// TIA Portal V19 export
FUNCTION_BLOCK "ValveMonitor"   // FB2, STL
TITLE = Valve Monitor
{ S7_Optimized_Access := 'TRUE' }
// Valve Monitor monitors single acting valves with Energiseed only or 
// De-energised 
// only or both Feedback states. Selection of feedback states in use can be 
// selected with Bits 0 and 1 of the "ControlWord" Input.
// 
// 
// Control Word
// Bit 0 = IN_DE in use
// Bit 1 = IN_EN in use
// 
// 
// Valve Monitor should be called within a Timed Interrupt OB and the duration 
// counters should be multiplied by the Timed Interrupt Cycle time to get the 
// durations in Seconds.
// 
// Note: If Activation State changes before destination FeedBack is reached then 
// the Duration count is not moved to the Archive and therefore does not affect 
// the 
// average duration. (De)Activations Count(s) will be incremented
// stored: AutoNumber false, MemoryReserve 100
   VAR_INPUT
      IN_EN : Bool;
      IN_DE : Bool;
      IN_ACT : Bool;
      ControlWord : Word;
   END_VAR
   VAR_IN_OUT
      Info : "ValvesInfo_UDT";
   END_VAR
   VAR
      ActMem : Bool;
      DeActMem : Bool;
      ActDur : Bool;
      DeActDur : Bool;
      ActClearDurCount : Bool;
      DeActClearDurCount : Bool;
      FP_A : Bool;
      FP_D : Bool;
      FP_A_Pulse : Bool;
      FP_D_Pulse : Bool;
      SumAverage : DInt;
      CountAverage : Int;
      data : "ValveMonitor_UDT";
   END_VAR
   VAR_TEMP
      EN_In_Use : Bool;
      DE_In_Use : Bool;
   END_VAR
BEGIN

NETWORK
TITLE = 
      A     #ControlWord.%X0;
      =     #EN_In_Use;
      A     #ControlWord.%X1;
      =     #DE_In_Use;


NETWORK
TITLE = RESET ALL Info
      A     #Info.RESET;
      JCN   RST;
      L     0;
// Act
      T     #data.Activation.ActivationCounter;
      T     #data.Activation.StrokeDuration.count;
      T     #data.Activation.StrokeDuration.Archive.n1;
      T     #data.Activation.StrokeDuration.Archive.n2;
      T     #data.Activation.StrokeDuration.Archive.n3;
      T     #data.Activation.StrokeDuration.Archive.n4;
      T     #data.Activation.StrokeDuration.Archive.n5;
      T     #data.Activation.StrokeDuration.Archive.n6;
      T     #data.Activation.StrokeDuration.Archive.n7;
      T     #data.Activation.StrokeDuration.Archive.n8;
      T     #data.Activation.StrokeDuration.Archive.n9;
      T     #data.Activation.StrokeDuration.Archive.n10;
// De_Act
      T     #data.De_Activation.De_ActivationCounter;
      T     #data.De_Activation.StrokeDuration.count;
      T     #data.De_Activation.StrokeDuration.Archive.n1;
      T     #data.De_Activation.StrokeDuration.Archive.n2;
      T     #data.De_Activation.StrokeDuration.Archive.n3;
      T     #data.De_Activation.StrokeDuration.Archive.n4;
      T     #data.De_Activation.StrokeDuration.Archive.n5;
      T     #data.De_Activation.StrokeDuration.Archive.n6;
      T     #data.De_Activation.StrokeDuration.Archive.n7;
      T     #data.De_Activation.StrokeDuration.Archive.n8;
      T     #data.De_Activation.StrokeDuration.Archive.n9;
      T     #data.De_Activation.StrokeDuration.Archive.n10;
      R     #Info.RESET;
RST:  NOP   0;


NETWORK
TITLE = Activation Counter
      A     #IN_ACT;
      AN    #IN_EN;
      AN    #ActMem;
      S     #ActMem;
      R     #DeActMem;

      A     #ActMem;
      FP    #FP_A;
      =     #FP_A_Pulse;
      JCN   ACTC;
      L     #data.Activation.ActivationCounter;
      L     1;
      +I;
      T     #data.Activation.ActivationCounter;
ACTC: NOP   0;


NETWORK
TITLE = De-Activation Counter
      AN    #IN_ACT;
      AN    #IN_DE;
      AN    #DeActMem;
      S     #DeActMem;
      R     #ActMem;

      A     #DeActMem;
      FP    #FP_D;
      =     #FP_D_Pulse;
      JCN   DACC;
      L     #data.De_Activation.De_ActivationCounter;
      L     1;
      +I;
      T     #data.De_Activation.De_ActivationCounter;
DACC: NOP   0;



NETWORK
TITLE = Activation Duration
      A     #EN_In_Use;  // IN_EN in Use
      JCN   ENDA;  // Jump to ENDA if False
      A     #FP_A_Pulse;
      AN    #IN_EN;
      S     #ActDur;

      A     #ActDur;
      A     #IN_EN;
      ON    #IN_ACT;
      R     #ActDur;
      R     #ActClearDurCount;
// Move Duration Count to Archive.n1
      AN    #ActDur;
      A     #IN_ACT;
      JCN   MOV;
      L     #data.Activation.StrokeDuration.count;
      T     #data.Activation.StrokeDuration.Archive.n1;
MOV:  NOP   0;

//Clear Counter
      A     #ActDur;
      AN    #ActClearDurCount;
      JCN   ATCC;
      L     0;
      T     #data.Activation.StrokeDuration.count;
      SET;
      S     #ActClearDurCount;
// Shift Archive data
      L     #data.Activation.StrokeDuration.Archive.n9;
      T     #data.Activation.StrokeDuration.Archive.n10;
      L     #data.Activation.StrokeDuration.Archive.n8;
      T     #data.Activation.StrokeDuration.Archive.n9;
      L     #data.Activation.StrokeDuration.Archive.n7;
      T     #data.Activation.StrokeDuration.Archive.n8;
      L     #data.Activation.StrokeDuration.Archive.n6;
      T     #data.Activation.StrokeDuration.Archive.n7;
      L     #data.Activation.StrokeDuration.Archive.n5;
      T     #data.Activation.StrokeDuration.Archive.n6;
      L     #data.Activation.StrokeDuration.Archive.n4;
      T     #data.Activation.StrokeDuration.Archive.n5;
      L     #data.Activation.StrokeDuration.Archive.n3;
      T     #data.Activation.StrokeDuration.Archive.n4;
      L     #data.Activation.StrokeDuration.Archive.n2;
      T     #data.Activation.StrokeDuration.Archive.n3;
      L     #data.Activation.StrokeDuration.Archive.n1;
      T     #data.Activation.StrokeDuration.Archive.n2;
ATCC: NOP   0;

// Count Duration
      A     #ActDur;
      A     #ActClearDurCount;
      JCN   _0CD;
      L     #data.Activation.StrokeDuration.count;
      L     1;
      +I;
      T     #data.Activation.StrokeDuration.count;
_0CD: NOP   0;
ENDA: NOP   0;




NETWORK
TITLE = DeDeActivation Duration
      A     #DE_In_Use;  // IN_DE in Use
      JCN   ENDD;  // Jump to ENDA if False
      A     #FP_D_Pulse;
      AN    #IN_DE;
      S     #DeActDur;

      A     #DeActDur;
      A     #IN_DE;
      O     #IN_ACT;
      R     #DeActDur;
      R     #DeActClearDurCount;
// Move Duration Count to Archive.n1
      AN    #DeActDur;
      AN    #IN_ACT;
      JCN   MOVD;
      L     #data.De_Activation.StrokeDuration.count;
      T     #data.De_Activation.StrokeDuration.Archive.n1;
MOVD: NOP   0;

//Clear Counter
      A     #DeActDur;
      AN    #DeActClearDurCount;
      JCN   DTCC;
      L     0;
      T     #data.De_Activation.StrokeDuration.count;
      SET;
      S     #DeActClearDurCount;
// Shift Archive data
      L     #data.De_Activation.StrokeDuration.Archive.n9;
      T     #data.De_Activation.StrokeDuration.Archive.n10;
      L     #data.De_Activation.StrokeDuration.Archive.n8;
      T     #data.De_Activation.StrokeDuration.Archive.n9;
      L     #data.De_Activation.StrokeDuration.Archive.n7;
      T     #data.De_Activation.StrokeDuration.Archive.n8;
      L     #data.De_Activation.StrokeDuration.Archive.n6;
      T     #data.De_Activation.StrokeDuration.Archive.n7;
      L     #data.De_Activation.StrokeDuration.Archive.n5;
      T     #data.De_Activation.StrokeDuration.Archive.n6;
      L     #data.De_Activation.StrokeDuration.Archive.n4;
      T     #data.De_Activation.StrokeDuration.Archive.n5;
      L     #data.De_Activation.StrokeDuration.Archive.n3;
      T     #data.De_Activation.StrokeDuration.Archive.n4;
      L     #data.De_Activation.StrokeDuration.Archive.n2;
      T     #data.De_Activation.StrokeDuration.Archive.n3;
      L     #data.De_Activation.StrokeDuration.Archive.n1;
      T     #data.De_Activation.StrokeDuration.Archive.n2;
DTCC: NOP   0;

// Count Duration
      A     #DeActDur;
      A     #DeActClearDurCount;
      JCN   D0CD;
      L     #data.De_Activation.StrokeDuration.count;
      L     1;
      +I;
      T     #data.De_Activation.StrokeDuration.count;
D0CD: NOP   0;
ENDD: NOP   0;




NETWORK
TITLE = Average Activation Duration Count
      L     0;
      T     #SumAverage;
      T     #CountAverage;


      L     #data.Activation.StrokeDuration.Archive.n1;
      L     0;
      >I;
      JCN   a001;
      L     1;
      L     #CountAverage;
      +I;
      T     #CountAverage;
      L     #data.Activation.StrokeDuration.Archive.n1;
      L     #SumAverage;
      +I;
      T     #SumAverage;
a001: L     #data.Activation.StrokeDuration.Archive.n2;
      L     0;
      >I;
      JCN   a002;
      L     1;
      L     #CountAverage;
      +I;
      T     #CountAverage;
      L     #data.Activation.StrokeDuration.Archive.n2;
      L     #SumAverage;
      +I;
      T     #SumAverage;
a002: L     #data.Activation.StrokeDuration.Archive.n3;
      L     0;
      >I;
      JCN   a003;
      L     1;
      L     #CountAverage;
      +I;
      T     #CountAverage;
      L     #data.Activation.StrokeDuration.Archive.n3;
      L     #SumAverage;
      +I;
      T     #SumAverage;
a003: L     #data.Activation.StrokeDuration.Archive.n4;
      L     0;
      >I;
      JCN   a004;
      L     1;
      L     #CountAverage;
      +I;
      T     #CountAverage;
      L     #data.Activation.StrokeDuration.Archive.n4;
      L     #SumAverage;
      +I;
      T     #SumAverage;
a004: L     #data.Activation.StrokeDuration.Archive.n5;
      L     0;
      >I;
      JCN   a005;
      L     1;
      L     #CountAverage;
      +I;
      T     #CountAverage;
      L     #data.Activation.StrokeDuration.Archive.n5;
      L     #SumAverage;
      +I;
      T     #SumAverage;
a005: L     #data.Activation.StrokeDuration.Archive.n6;
      L     0;
      >I;
      JCN   a006;
      L     1;
      L     #CountAverage;
      +I;
      T     #CountAverage;
      L     #data.Activation.StrokeDuration.Archive.n6;
      L     #SumAverage;
      +I;
      T     #SumAverage;
a006: L     #data.Activation.StrokeDuration.Archive.n7;
      L     0;
      >I;
      JCN   a007;
      L     1;
      L     #CountAverage;
      +I;
      T     #CountAverage;
      L     #data.Activation.StrokeDuration.Archive.n7;
      L     #SumAverage;
      +I;
      T     #SumAverage;
a007: L     #data.Activation.StrokeDuration.Archive.n8;
      L     0;
      >I;
      JCN   a008;
      L     1;
      L     #CountAverage;
      +I;
      T     #CountAverage;
      L     #data.Activation.StrokeDuration.Archive.n8;
      L     #SumAverage;
      +I;
      T     #SumAverage;
a008: L     #data.Activation.StrokeDuration.Archive.n9;
      L     0;
      >I;
      JCN   a009;
      L     1;
      L     #CountAverage;
      +I;
      T     #CountAverage;
      L     #data.Activation.StrokeDuration.Archive.n9;
      L     #SumAverage;
      +I;
      T     #SumAverage;
a009: L     #data.Activation.StrokeDuration.Archive.n10;
      L     0;
      >I;
      JCN   a010;
      L     1;
      L     #CountAverage;
      +I;
      T     #CountAverage;
      L     #data.Activation.StrokeDuration.Archive.n10;
      L     #SumAverage;
      +I;
      T     #SumAverage;
a010: NOP   0;
// Calculate Average
      L     #SumAverage;
      L     #CountAverage;
      /D;
      T     #data.Activation.StrokeDuration.Average;


NETWORK
TITLE = Average De_Activation Duration Count
      L     0;
      T     #SumAverage;
      T     #CountAverage;


      L     #data.Activation.StrokeDuration.Archive.n1;
      L     0;
      >I;
      JCN   d001;
      L     1;
      L     #CountAverage;
      +I;
      T     #CountAverage;
      L     #data.De_Activation.StrokeDuration.Archive.n1;
      L     #SumAverage;
      +I;
      T     #SumAverage;
d001: L     #data.De_Activation.StrokeDuration.Archive.n2;
      L     0;
      >I;
      JCN   d002;
      L     1;
      L     #CountAverage;
      +I;
      T     #CountAverage;
      L     #data.De_Activation.StrokeDuration.Archive.n2;
      L     #SumAverage;
      +I;
      T     #SumAverage;
d002: L     #data.De_Activation.StrokeDuration.Archive.n3;
      L     0;
      >I;
      JCN   d003;
      L     1;
      L     #CountAverage;
      +I;
      T     #CountAverage;
      L     #data.De_Activation.StrokeDuration.Archive.n3;
      L     #SumAverage;
      +I;
      T     #SumAverage;
d003: L     #data.De_Activation.StrokeDuration.Archive.n4;
      L     0;
      >I;
      JCN   d004;
      L     1;
      L     #CountAverage;
      +I;
      T     #CountAverage;
      L     #data.De_Activation.StrokeDuration.Archive.n4;
      L     #SumAverage;
      +I;
      T     #SumAverage;
d004: L     #data.De_Activation.StrokeDuration.Archive.n5;
      L     0;
      >I;
      JCN   d005;
      L     1;
      L     #CountAverage;
      +I;
      T     #CountAverage;
      L     #data.De_Activation.StrokeDuration.Archive.n5;
      L     #SumAverage;
      +I;
      T     #SumAverage;
d005: L     #data.De_Activation.StrokeDuration.Archive.n6;
      L     0;
      >I;
      JCN   d006;
      L     1;
      L     #CountAverage;
      +I;
      T     #CountAverage;
      L     #data.De_Activation.StrokeDuration.Archive.n6;
      L     #SumAverage;
      +I;
      T     #SumAverage;
d006: L     #data.De_Activation.StrokeDuration.Archive.n7;
      L     0;
      >I;
      JCN   d007;
      L     1;
      L     #CountAverage;
      +I;
      T     #CountAverage;
      L     #data.De_Activation.StrokeDuration.Archive.n7;
      L     #SumAverage;
      +I;
      T     #SumAverage;
d007: L     #data.De_Activation.StrokeDuration.Archive.n8;
      L     0;
      >I;
      JCN   d008;
      L     1;
      L     #CountAverage;
      +I;
      T     #CountAverage;
      L     #data.De_Activation.StrokeDuration.Archive.n8;
      L     #SumAverage;
      +I;
      T     #SumAverage;
d008: L     #data.De_Activation.StrokeDuration.Archive.n9;
      L     0;
      >I;
      JCN   d009;
      L     1;
      L     #CountAverage;
      +I;
      T     #CountAverage;
      L     #data.De_Activation.StrokeDuration.Archive.n9;
      L     #SumAverage;
      +I;
      T     #SumAverage;
d009: L     #data.De_Activation.StrokeDuration.Archive.n10;
      L     0;
      >I;
      JCN   d010;
      L     1;
      L     #CountAverage;
      +I;
      T     #CountAverage;
      L     #data.De_Activation.StrokeDuration.Archive.n10;
      L     #SumAverage;
      +I;
      T     #SumAverage;
d010: NOP   0;
// Calculate Average
      L     #SumAverage;
      L     #CountAverage;
      /D;
      T     #data.De_Activation.StrokeDuration.Average;


NETWORK
TITLE = Move Data to Out Info
      L     #data.Activation.ActivationCounter;
      T     #Info.Act.Count;
      L     #data.Activation.StrokeDuration.count;
      T     #Info.Act.Duration;
      L     #data.Activation.StrokeDuration.Average;
      T     #Info.Act.AvgDuration;

      L     #data.De_Activation.De_ActivationCounter;
      T     #Info.DeAct.Count;
      L     #data.De_Activation.StrokeDuration.count;
      T     #Info.DeAct.Duration;
      L     #data.De_Activation.StrokeDuration.Average;
      T     #Info.DeAct.AvgDuration;



END_FUNCTION_BLOCK
